PROGRAM HMI_Ultimate_Limit
VAR
	DownUltLimit: DWORD;
END_VAR

IF GV_Lift.ULTIMATE_LIMIT_INDICATOR_OUT THEN
	DownUltLimit := GV_HMI.dwRed;
ELSIF GV_Lift.ULTIMATE_LIMIT_INDICATOR_LATCH_OUT THEN
	DownUltLimit := GV_HMI.dwYellow;
ELSE DownUltLimit := GV_HMI.dwGreen;
END_IF

END_PROGRAM

(* stored: Version 1.1.0.1, ProductVersion 3.1.4022.12
   POU HMI_Ultimate_Limit: Id {1bd66aa5-721b-45f5-9953-10e6f1eb9311}, SpecialFunc None *)
